TYPE ST_SZ_Zustand :
STRUCT
	Arbeit						: REAL;
	Freigabe					: BOOL;
	Leistung					: REAL;
	Leistungsfaktor				: REAL;


END_STRUCT
END_TYPE

(* stored: Version 1.1.0.1, ProductVersion 3.1.4024.9
   DUT ST_SZ_Zustand: Id {fdba494e-6c99-4e4a-9148-466b927dc2ed} *)
